// TIA Portal V20 export
TYPE "LER_typeServoTorqueCalInterface"
// stored: Access Published
   STRUCT
      commands : "LER_typeServoTorqueCalCommands";
      monitoring : "LER_typeServoTorqueCalMonitoring";
   END_STRUCT;
END_TYPE
